// TwinCAT 3 PLC project Untitled1
// ProgramVersion: 3.1.4024.0
// libraries:
//   Tc2_Standard, * (Beckhoff Automation GmbH)
//   Tc2_System, * (Beckhoff Automation GmbH)
//   Tc3_Module, * (Beckhoff Automation GmbH)
// project tree:
//   GVLs/ MachineObjectsArray.TcGVL
//   / PlcTask.TcTTO
//   POUs/ FB_SafetyTestTrolley.TcPOU, MAIN.TcPOU
// real-time tasks:
//   TASK PlcTask: cycle T#10ms, priority 20, ADS port 350
// I/O:
//   DEVICE Device 1 (EtherCAT) (disabled), AmsNetId 10.100.30.103.2.1
//     Term 1 (EK1100) [EK1100 EtherCAT Coupler (2A E-Bus)]
//       Term 2 (EL2008) [EL2008 8Ch. Dig. Output 24V, 0.5A]
//       Term 3 (EL1008) [EL1008 8Ch. Dig. Input 24V, 3ms]

CONFIGURATION Untitled1
    RESOURCE PLC ON TwinCAT3
        TASK PlcTask(INTERVAL := T#10ms, PRIORITY := 20);
        PROGRAM MAIN WITH PlcTask : MAIN;
    END_RESOURCE
END_CONFIGURATION

// ---- GVLs/MachineObjectsArray.TcGVL
// Upper bounds of devices
VAR_GLOBAL CONSTANT
    cUpperBoundSafetyTestTrolley    : UINT := 4;
END_VAR

VAR_GLOBAL
    {attribute 'TcContextName':='MainTask'}
    SafetyTestTrolley   : ARRAY [0..cUpperBoundSafetyTestTrolley] OF FB_SafetyTestTrolley;
END_VAR

// ---- POUs/MAIN.TcPOU
PROGRAM MAIN
VAR
END_VAR

END_PROGRAM

// ---- POUs/FB_SafetyTestTrolley.TcPOU
FUNCTION_BLOCK FB_SafetyTestTrolley
VAR_INPUT
    // Transportsystem
    // Lamp Reset Buttons
    arrLampResetButtons_TS      AT%I*    : ARRAY [0..7] OF BOOL;
    
    // Emergency Stop Buttons
    arrEmergencyStopButtons_TS  AT%Q*    : ARRAY [0..7] OF BOOL;
    
    // Reset Buttons
    arrResetButtons_TS          AT%Q*    : ARRAY [0..7] OF BOOL;
    
    // Lightcurtains
    arrLightcurtains_TS         AT%Q*    : ARRAY [0..7] OF BOOL;
    
    // Interlocking Guards
    arrInterlockingGuards_TS    AT%Q*    : ARRAY [0..3] OF BOOL;

    // Machinezone
    // Lamp Reset Button
    bLampResetButton1_MZ        AT%I*   : BOOL;
    // Emergency Stop Button
    bEmergencyStopButton1_MZ    AT%Q*   : BOOL;
    // Reset Button
    bResetButton1_MZ            AT%Q*   : BOOL;
    // Lightcurtain
    bLightcurtain1_MZ           AT%Q*   : BOOL;
    // Interlocking Guard
    bInterlockingGuard1_MZ      AT%Q*   : BOOL;
END_VAR

END_FUNCTION_BLOCK
